/// Implicitly generated code : DO NOT EDIT
/// Checks for division by 0, if divisor is 0, replace it with 1 and report error
{attribute 'check_div_real32' := ''}
{attribute 'no_check' := ''}
FUNCTION CheckDivReal : REAL
VAR_INPUT
	divisor: REAL;
END_VAR

IF divisor = 0 THEN
	// replace divisor and report error if necessary
	CheckDivReal := 1;
	GVL_Supervision.aCodeErr[eCodeError_divReal] := TRUE;
ELSE
	CheckDivReal := divisor;
END_IF;

END_FUNCTION

(* stored: Version 1.1.0.1, ProductVersion 3.1.4022.9
   POU CheckDivReal: Id {e786fb56-4b1e-4276-b1e0-de740d9650ce}, SpecialFunc None *)
